// TIA Portal V20 export
FUNCTION_BLOCK "LER_EQP_Interface_ReelCut"   // FB129, LAD
// stored: Access Published, MemoryReserve 100, SetENOAutomatically false
   VAR_INPUT
      enable : Bool;
      executeCmd : Bool;
      clock : Bool;
      heartBeat : Byte;
      unitStatus : "LAF_typeUnitStatus";
      unitAlarms : "LAF_typeAlarms";
   END_VAR
   VAR_OUTPUT
      error : Bool;
      status : Word;
   END_VAR
   VAR_IN_OUT
      reelcutCommunication : "LER_typeCommunicationReelCut";
      configuration : "LER_typeCommunicationConfiguration";
      moduleInterface : "LER_typeCommunicationInterface";
      controlNode : "LER_typeCommunicationControlNode";
   END_VAR
   VAR
      instEQP_Interface_Communication { S7_SetPoint := 'True'} : "LER_EQP_Communication";
      statReelCutHeartBeat : Byte;
      statStackState : Struct
         Stop : Bool;
         Abort : Bool;
         Hold : Bool;
         Complete : Bool;
         Idle : Bool;
         TotalStop : Bool;
      END_STRUCT;
      statTonTimer : Array[0..9] of TON_TIME;
      statTofTimer : Array[0..9] of TOF_TIME;
   END_VAR
   VAR CONSTANT
      STATUS_NO_ERROR_OCCURRED : Word := 16#0;
      ERR_HEARTBEAT_ERROR : Word := 16#8000;
   END_VAR
BEGIN

REGION Network 1: EQP Interface Stack State
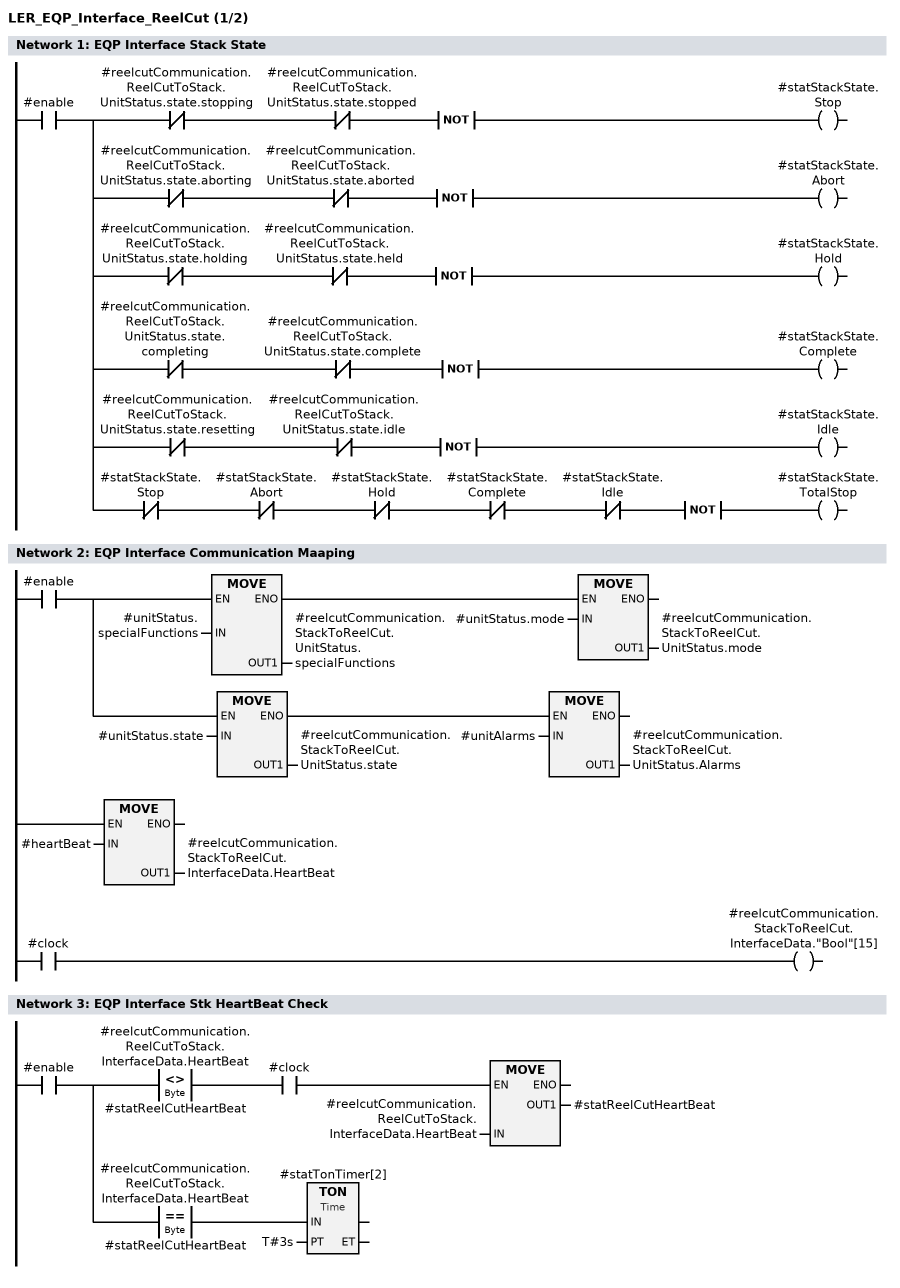
   RUNG wire#powerrail
      Contact( #enable )
      wire#w1
      I_Contact( #reelcutCommunication.ReelCutToStack.UnitStatus.state.stopping )
      I_Contact( #reelcutCommunication.ReelCutToStack.UnitStatus.state.stopped )
      Not()
      Coil( #statStackState.Stop )
   END_RUNG
   RUNG wire#w1
      I_Contact( #reelcutCommunication.ReelCutToStack.UnitStatus.state.aborting )
      I_Contact( #reelcutCommunication.ReelCutToStack.UnitStatus.state.aborted )
      Not()
      Coil( #statStackState.Abort )
   END_RUNG
   RUNG wire#w1
      I_Contact( #reelcutCommunication.ReelCutToStack.UnitStatus.state.holding )
      I_Contact( #reelcutCommunication.ReelCutToStack.UnitStatus.state.held )
      Not()
      Coil( #statStackState.Hold )
   END_RUNG
   RUNG wire#w1
      I_Contact( #reelcutCommunication.ReelCutToStack.UnitStatus.state.completing )
      I_Contact( #reelcutCommunication.ReelCutToStack.UnitStatus.state.complete )
      Not()
      Coil( #statStackState.Complete )
   END_RUNG
   RUNG wire#w1
      I_Contact( #reelcutCommunication.ReelCutToStack.UnitStatus.state.resetting )
      I_Contact( #reelcutCommunication.ReelCutToStack.UnitStatus.state.idle )
      Not()
      Coil( #statStackState.Idle )
   END_RUNG
   RUNG wire#w1
      I_Contact( #statStackState.Stop )
      I_Contact( #statStackState.Abort )
      I_Contact( #statStackState.Hold )
      I_Contact( #statStackState.Complete )
      I_Contact( #statStackState.Idle )
      Not()
      Coil( #statStackState.TotalStop )
   END_RUNG
   // the same network as SCL:
   #statStackState.Stop := NOT (#enable AND NOT #reelcutCommunication.ReelCutToStack.UnitStatus.state.stopping AND NOT #reelcutCommunication.ReelCutToStack.UnitStatus.state.stopped);
   #statStackState.Abort := NOT (#enable AND NOT #reelcutCommunication.ReelCutToStack.UnitStatus.state.aborting AND NOT #reelcutCommunication.ReelCutToStack.UnitStatus.state.aborted);
   #statStackState.Hold := NOT (#enable AND NOT #reelcutCommunication.ReelCutToStack.UnitStatus.state.holding AND NOT #reelcutCommunication.ReelCutToStack.UnitStatus.state.held);
   #statStackState.Complete := NOT (#enable AND NOT #reelcutCommunication.ReelCutToStack.UnitStatus.state.completing AND NOT #reelcutCommunication.ReelCutToStack.UnitStatus.state.complete);
   #statStackState.Idle := NOT (#enable AND NOT #reelcutCommunication.ReelCutToStack.UnitStatus.state.resetting AND NOT #reelcutCommunication.ReelCutToStack.UnitStatus.state.idle);
   #statStackState.TotalStop := NOT (#enable AND NOT #statStackState.Stop AND NOT #statStackState.Abort AND NOT #statStackState.Hold AND NOT #statStackState.Complete AND NOT #statStackState.Idle);
END_REGION

REGION Network 2: EQP Interface Communication Maaping
   RUNG wire#powerrail
      Contact( #enable )
      wire#w1
      Move(in := #unitStatus.specialFunctions, out1 => #reelcutCommunication.StackToReelCut.UnitStatus.specialFunctions)
      Move(in := #unitStatus.mode, out1 => #reelcutCommunication.StackToReelCut.UnitStatus.mode)
   END_RUNG
   RUNG wire#w1
      Move(in := #unitStatus.state, out1 => #reelcutCommunication.StackToReelCut.UnitStatus.state)
      Move(in := #unitAlarms, out1 => #reelcutCommunication.StackToReelCut.UnitStatus.Alarms)
   END_RUNG
   RUNG wire#powerrail
      Move(in := #heartBeat, out1 => #reelcutCommunication.StackToReelCut.InterfaceData.HeartBeat)
   END_RUNG
   RUNG wire#powerrail
      Contact( #clock )
      Coil( #reelcutCommunication.StackToReelCut.InterfaceData."Bool"[15] )
   END_RUNG
   // the same network as SCL:
   IF #enable THEN
       #reelcutCommunication.StackToReelCut.UnitStatus.specialFunctions := #unitStatus.specialFunctions;
       #reelcutCommunication.StackToReelCut.UnitStatus.mode := #unitStatus.mode;
       #reelcutCommunication.StackToReelCut.UnitStatus.state := #unitStatus.state;
       #reelcutCommunication.StackToReelCut.UnitStatus.Alarms := #unitAlarms;
   END_IF;
   #reelcutCommunication.StackToReelCut.InterfaceData.HeartBeat := #heartBeat;
   #reelcutCommunication.StackToReelCut.InterfaceData."Bool"[15] := #clock;
END_REGION

REGION Network 3: EQP Interface Stk HeartBeat Check
   RUNG wire#powerrail
      Contact( #enable )
      wire#w1
      { S7_Templates := "SrcType := Byte" } NE_Contact(in1 := #reelcutCommunication.ReelCutToStack.InterfaceData.HeartBeat, in2 := #statReelCutHeartBeat)
      Contact( #clock )
      Move(in := #reelcutCommunication.ReelCutToStack.InterfaceData.HeartBeat, out1 => #statReelCutHeartBeat)
   END_RUNG
   RUNG wire#w1
      { S7_Templates := "SrcType := Byte" } EQ_Contact(in1 := #reelcutCommunication.ReelCutToStack.InterfaceData.HeartBeat, in2 := #statReelCutHeartBeat)
      { S7_Templates := "time_type := Time" } #statTonTimer[2].TON(pt := T#3s, et =>)
   END_RUNG
   // the same network as SCL:
   IF #enable AND (#reelcutCommunication.ReelCutToStack.InterfaceData.HeartBeat <> #statReelCutHeartBeat) AND #clock THEN
       #statReelCutHeartBeat := #reelcutCommunication.ReelCutToStack.InterfaceData.HeartBeat;
   END_IF;
   #statTonTimer[2].TON(IN := #enable AND (#reelcutCommunication.ReelCutToStack.InterfaceData.HeartBeat = #statReelCutHeartBeat),
                        PT := T#3s);
END_REGION

REGION Network 4: EQP Interface Communication Stack <-> ReelCut
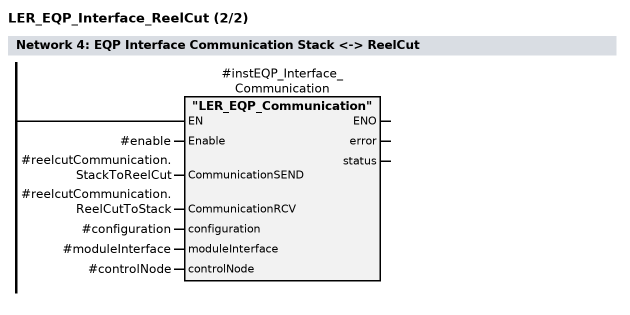
   RUNG wire#powerrail
      #instEQP_Interface_Communication(Enable := #enable, CommunicationSEND := #reelcutCommunication.StackToReelCut, CommunicationRCV := #reelcutCommunication.ReelCutToStack, configuration := #configuration, moduleInterface := #moduleInterface, controlNode := #controlNode, error =>, status =>)
   END_RUNG
   // the same network as SCL:
   #instEQP_Interface_Communication(Enable := #enable,   // "LER_EQP_Communication"
                           CommunicationSEND := #reelcutCommunication.StackToReelCut,
                           CommunicationRCV := #reelcutCommunication.ReelCutToStack,
                           configuration := #configuration,
                           moduleInterface := #moduleInterface,
                           controlNode := #controlNode);
END_REGION

REGION Network 5 (SCL): Error Check
   REGION Error Code Search

       IF #enable AND NOT #configuration.disableAlarms THEN
           IF #statTonTimer[2].Q THEN
               #status := #ERR_HEARTBEAT_ERROR;

           ELSIF #instEQP_Interface_Communication.error THEN
               #status := #instEQP_Interface_Communication.status;

           ELSE
               #status := #STATUS_NO_ERROR_OCCURRED;

           END_IF;
       ELSE
           #status := #STATUS_NO_ERROR_OCCURRED;

       END_IF;


       // Error Bit
       #error := #status <> 0;

   END_REGION
END_REGION

REGION Network 6 (SCL): ##### Outputs mapping #####
   #moduleInterface.monitoring.error := #error;
   #moduleInterface.monitoring.status := #status;

   #controlNode.monitoring := #moduleInterface.monitoring;
END_REGION
END_FUNCTION_BLOCK
